FUNCTION_BLOCK controller (* ODE *)
  (* Standard: 61499-2 *)
  (* Version 0.1, 2017-00-25, hpea485, UOA *)
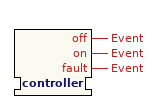
  EVENT_OUTPUT
    off;
    on;
    fault;
  END_EVENT
  VAR
    StateChangeTime : LREAL := 5.0;
    DeltaTime : LREAL := 0.01;
    x : LREAL := 0;
  END_VAR
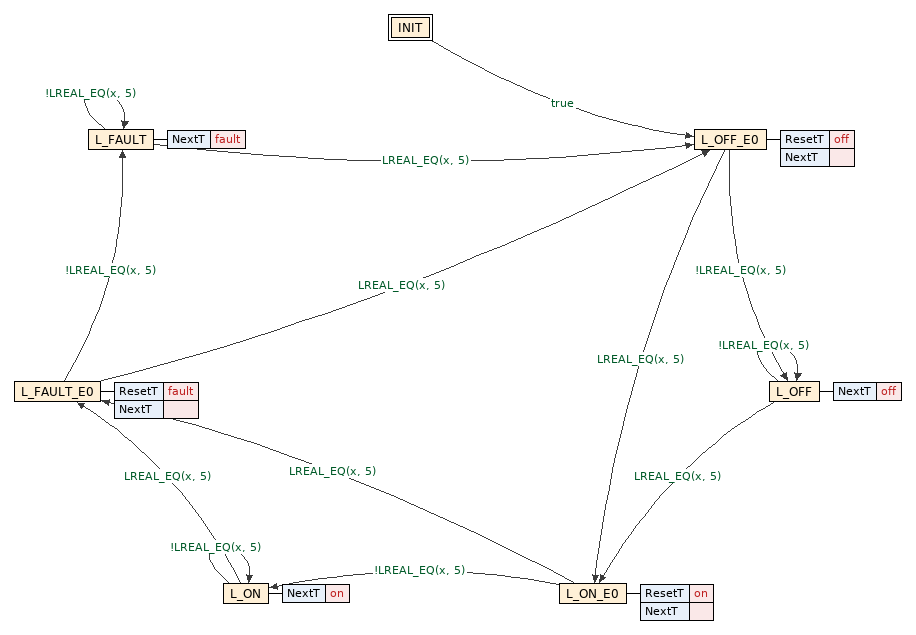
  EC_STATES
    INIT;
    L_OFF_E0 : ResetT -> off, NextT;
    L_OFF : NextT -> off;
    L_ON_E0 : ResetT -> on, NextT;
    L_ON : NextT -> on;
    L_FAULT_E0 : ResetT -> fault, NextT;
    L_FAULT : NextT -> fault;
  END_STATES
  EC_TRANSITIONS
    INIT TO L_OFF_E0 := true;
    L_OFF_E0 TO L_OFF := !LREAL_EQ(x, 5);
    L_OFF_E0 TO L_ON_E0 := LREAL_EQ(x, 5);
    L_OFF TO L_OFF := !LREAL_EQ(x, 5);
    L_OFF TO L_ON_E0 := LREAL_EQ(x, 5);
    L_ON_E0 TO L_ON := !LREAL_EQ(x, 5);
    L_ON_E0 TO L_FAULT_E0 := LREAL_EQ(x, 5);
    L_ON TO L_ON := !LREAL_EQ(x, 5);
    L_ON TO L_FAULT_E0 := LREAL_EQ(x, 5);
    L_FAULT_E0 TO L_FAULT := !LREAL_EQ(x, 5);
    L_FAULT_E0 TO L_OFF_E0 := LREAL_EQ(x, 5);
    L_FAULT TO L_FAULT := !LREAL_EQ(x, 5);
    L_FAULT TO L_OFF_E0 := LREAL_EQ(x, 5);
  END_TRANSITIONS
  ALGORITHM ResetT IN C: (* ODE_init *)
x_prime = 0;
  END_ALGORITHM
  ALGORITHM NextT IN C: (* ODE *)
x_dot = 1;
x_trigger = 5;
  END_ALGORITHM
END_FUNCTION_BLOCK
